{attribute 'qualified_only'}
{attribute 'strict'}
TYPE E_SocketSendState :
(
	READY,
	PREPARE_DATA,
	SENDING,
	AWAIT_RESPONSE,
	DONE,
	ERROR
);
END_TYPE

(* stored: Version 1.1.0.1, ProductVersion 3.1.4024.13
   DUT E_SocketSendState: Id {9fd162bf-4b85-4e67-b08a-b3574aa9ed3d} *)
